Fanuc TP program (LS listing): SIM_P_AND_P.LS

/PROG  SIM_P_AND_P
/ATTR
OWNER		= MNEDITOR;
COMMENT		= "";
PROG_SIZE	= 245;
CREATE		= DATE 25-11-12  TIME 15:30:52;
MODIFIED	= DATE 31-01-14  TIME 09:01:22;
FILE_NAME	= ;
VERSION		= 0;
LINE_COUNT	= 4;
MEMORY_SIZE	= 625;
PROTECT		= READ_WRITE;
TCD:  STACK_SIZE	= 0,
      TASK_PRIORITY	= 50,
      TIME_SLICE	= 0,
      BUSY_LAMP_OFF	= 0,
      ABORT_REQUEST	= 0,
      PAUSE_REQUEST	= 0;
DEFAULT_GROUP	= 1,*,*,*,*;
CONTROL_CODE	= 00000000 00000000;
/APPL
/APPL

AUTO_SINGULARITY_HEADER;
  ENABLE_SINGULARITY_AVOIDANCE   : TRUE;
/MN
   1:  CALL HANDOFF_SMPL    ;
   2:  CALL LUL_GRINDER_SMPL    ;
   3:  CALL HOME    ;
   4:  RO[1:Vacuum ON 1]=OFF ;
/POS
/END
